(* IEC 61131-3 sources: Masterarbeit-LP/openplc, 1 file *)

(* ---- testprogramm.st ---- *)
PROGRAM testprogramm
  VAR
    startsensor_1 AT %IX100.0 : BOOL;
    endsensor_1 AT %IX100.1 : BOOL;
    antrieb_1 AT %QX100.0 : BOOL;
    startsensor_2 AT %IX100.2 : BOOL;
    endsensor_2 AT %IX100.3 : BOOL;
    antrieb_2 AT %QX100.1 : BOOL;
    startsensor_3 AT %IX100.4 : BOOL;
    antrieb_3 AT %QX100.2 : BOOL;
  END_VAR
  VAR
    SR0 : SR;
    SR1 : SR;
    SR2 : SR;
  END_VAR
  VAR
    newantrieb AT %QX100.3 : BOOL;
    newsensor AT %IX100.6 : BOOL;
    palettedrinnen AT %IX100.7 : BOOL;
    gedreht AT %IX101.0 : BOOL;
    dreher AT %QX100.4 : BOOL;
    rfid AT %QX100.5 : BOOL;
    rfid2 AT %QX100.6 : BOOL;
    trigger_rfid AT %IX100.5 : BOOL;
    secondtrigger AT %IX101.1 : BOOL;
  END_VAR
  VAR
    TON0 : TON;
    delay : TIME := T#1s;
    currenttime : TIME := T#0s;
  END_VAR
  VAR
    direction AT %QW100 : INT;
  END_VAR
  VAR
    controlvalue : INT := 1;
  END_VAR
  VAR
    derwert AT %IW100 : INT;
  END_VAR
  VAR
    SR3 : SR;
  END_VAR
  VAR
    ende1 AT %IX101.2 : BOOL;
    ende2 AT %IX101.3 : BOOL;
  END_VAR
  VAR
    OR53_OUT : BOOL;
    EQ13_OUT : BOOL;
    NOT55_OUT : BOOL;
    AND16_OUT : BOOL;
    OR54_OUT : BOOL;
    EQ41_OUT : BOOL;
    AND17_OUT : BOOL;
  END_VAR

  SR0(S1 := startsensor_1, R := endsensor_1);
  antrieb_1 := SR0.Q1;
  OR53_OUT := OR(gedreht, secondtrigger);
  EQ13_OUT := EQ(derwert, controlvalue);
  NOT55_OUT := NOT(gedreht);
  AND16_OUT := AND(newsensor, EQ13_OUT, NOT55_OUT);
  OR54_OUT := OR(AND16_OUT, ende1, ende2);
  SR3(S1 := OR53_OUT, R := OR54_OUT);
  newantrieb := SR3.Q1;
  SR1(S1 := startsensor_2, R := endsensor_2);
  antrieb_2 := SR1.Q1;
  TON0(IN := palettedrinnen, PT := delay);
  SR2(S1 := startsensor_3, R := TON0.Q);
  antrieb_3 := SR2.Q1;
  EQ41_OUT := EQ(derwert, controlvalue);
  AND17_OUT := AND(newsensor, EQ41_OUT);
  dreher := AND17_OUT;
  currenttime := TON0.ET;
END_PROGRAM

CONFIGURATION Config0

  RESOURCE Res0 ON PLC
    TASK task0(INTERVAL := T#20ms,PRIORITY := 0);
    PROGRAM instance0 WITH task0 : testprogramm;
  END_RESOURCE
END_CONFIGURATION
